// TIA Portal V19 export
DATA_BLOCK "LB114_FeedA01"   // DB125
// stored: InstanceOfName ButtonsSafe_LB114_FeedA01, InstanceOfType FB
"ButtonsSafe_LB114_FeedA01"
   // VAR_INPUT
   //    Reset_OthersPBs_Activation_IN : Bool;
   // END_VAR
   // VAR_OUTPUT
   //    Reset_OthersPBs_Activation_OUT : Bool;
   // END_VAR
   // VAR
   //    i : Int;
   //    iOperation : Int;
   //    iConcurrentOperation : Int;
   //    SettingWriteDone : Bool;
   //    PbPanel : "Buttons2Hands";
   //    PB : Struct
   //       ResetAlarms : Bool;
   //       Straightner_Fwd : Bool;
   //       Straightner_Bwd : Bool;
   //    END_STRUCT;
   // END_VAR
BEGIN
END_DATA_BLOCK
